PROGRAM BASE
VAR
	DateTime : FB_DATETIME;
	Strings : FB_STRINGS;
END_VAR

DateTime();
Strings();

END_PROGRAM

(* stored: Version 1.1.0.1, ProductVersion 3.1.4024.12
   POU BASE: Id {ff08221e-1d32-4986-8602-1c09f6f84525}, SpecialFunc None *)
